TYPE U_Simple :
UNION
	bMember  		: BOOL;
    dtMember 		: DT;
	nMember   		: DINT;
END_UNION
END_TYPE

(* stored: Version 1.1.0.1
   DUT U_Simple: Id {a50af2f4-50ec-4519-81e9-5e8da6a1620c} *)
